{attribute 'no_explicit_call' := 'do not call this function block directly'}
FUNCTION_BLOCK FB_Scalar IMPLEMENTS I_Scalar, I_Addition, I_Subtraction, I_Multiplication, I_Division
VAR
	_fValue : LREAL; 
END_VAR

METHOD DivideBy : I_Division
VAR_INPUT
	ipObject : I_Object;
END_VAR
VAR_OUTPUT
	e : E_OperatorError;
END_VAR
VAR
	Tmp : LREAL;
	ipNumber : I_Scalar;
END_VAR
DivideBy := THIS^;

IF NOT __QUERYINTERFACE(ipObject, ipNumber) THEN e := E_OperatorError.TypeMismatch; RETURN; END_IF

Tmp := ipNumber.ToF64(e => e);
IF Tmp = 0 THEN 
	THIS^._fValue := SEL(Tmp > 0, -1*TO_LREAL('#Inf'), TO_LREAL('#Inf'));
	RETURN;
	END_IF

IF e <> E_OperatorError.NoError THEN 
	THIS^._fValue := ipNumber.ToF64();
	END_IF

THIS^._fValue := THIS^.ToF64() / ipNumber.ToF64();
END_METHOD

{attribute 'hide'}
METHOD FB_init : BOOL
VAR_INPUT
	bInitRetains : BOOL; // if TRUE, the retain variables are initialized (warm start / cold start)
	bInCopyCode : BOOL;  // if TRUE, the instance afterwards gets moved into the copy code (online change)
	fInitValue : LREAL;
END_VAR
THIS^._fValue := fInitValue;
END_METHOD

METHOD Minus : I_Subtraction
VAR_INPUT
	ipObject : I_Object;
END_VAR
VAR_OUTPUT
	e : E_OperatorError;
END_VAR
VAR
	e1, e2 : E_OperatorError;
	ipNumber : I_Scalar;
END_VAR
Minus := THIS^;

IF NOT __QUERYINTERFACE(ipObject, ipNumber) THEN
  e := E_OperatorError.TypeMismatch; 
  RETURN;
  END_IF

THIS^._fValue := THIS^.ToF64(e => e1) - ipNumber.ToF64(e => e2);

e := MAX(e1, e2);
END_METHOD

METHOD Plus : I_Addition
VAR_INPUT
	ipObject : I_Object;
END_VAR
VAR_OUTPUT
	e : E_OperatorError;
END_VAR
VAR
	e1, e2 : E_OperatorError;
	ipNumber : I_Scalar;
END_VAR
Plus := THIS^;

IF NOT __QUERYINTERFACE(ipObject, ipNumber) THEN e := E_OperatorError.TypeMismatch; RETURN; END_IF

THIS^._fValue := THIS^.ToF64(e => e1) + ipNumber.ToF64(e => e2);

e := MAX(e1, e2);
END_METHOD

METHOD SetValue : REFERENCE TO FB_Scalar
VAR_INPUT
	fValue : LREAL;
END_VAR
SetValue REF= THIS^;

THIS^._fValue := fValue;
END_METHOD

METHOD Times : I_Multiplication
VAR_INPUT
	ipObject : I_Object;
END_VAR
VAR_OUTPUT
	e : E_OperatorError;
END_VAR
VAR
	e1, e2 : E_OperatorError;
	ipNumber : I_Scalar;
END_VAR
Times := THIS^;

IF NOT __QUERYINTERFACE(ipObject, ipNumber) THEN e := E_OperatorError.TypeMismatch; RETURN; END_IF

THIS^._fValue := THIS^.ToF64(e => e1) * ipNumber.ToF64( e => e2);

e := MAX(e1, e2);
END_METHOD

METHOD ToF64 : LREAL
VAR_OUTPUT
	e	: E_OperatorError;
END_VAR
ToF64 := THIS^._fValue;

IF TO_STRING(THIS^._fValue) = '#NaN' THEN 
	e := E_OperatorError.NaN;
ELSIF TO_STRING(THIS^._fValue) = '#Inf' THEN
	e := E_OperatorError.PositiveInfinity;
ELSIF TO_STRING(THIS^._fValue) = '-#Inf' THEN
	e := E_OperatorError.NegativeInfinity;
	END_IF
END_METHOD

METHOD ToI64 : LINT
VAR_OUTPUT
	e	: E_OperatorError;
END_VAR
ToI64 := TO_LINT(THIS^._fValue);

// Check for truncation.
IF Tc2_Math.FRAC(THIS^._fValue) <> 0  THEN 
	e := E_OperatorError.Truncation;
	END_IF
END_METHOD

METHOD ToU8 : BYTE
VAR_OUTPUT
	e	: E_OperatorError;
END_VAR
ToU8 := TO_BYTE(THIS^._fValue);

// Check for truncation.
IF Tc2_Math.FRAC(THIS^._fValue) <> 0  THEN 
	e := E_OperatorError.Truncation;
	END_IF

// Bounds check.
IF THIS^._fValue < 0 OR THIS^._fValue > 255 THEN 
	e := E_OperatorError.IntegerOverflow;
	END_IF
END_METHOD

END_FUNCTION_BLOCK

(* stored: Version 1.1.0.1, ProductVersion 3.1.4024.12
   POU FB_Scalar: Id {06260915-57c3-4c39-8ab5-e6a4c7e7c262}, SpecialFunc None
   Folder Constructor: Id {a996651f-3295-46b6-b977-e378ab8cc6d3}
   Folder IOperatorX: Id {fb9cacd6-caa0-492a-82b5-8880a839455e}
   Folder IScalar: Id {3e8f876f-10c8-4aaa-9fa8-9b178ddb88f2}
   Method DivideBy: Id {b0d0123e-cfb1-4101-8e18-a861c0279c74}
   Method FB_init: Id {63985488-ffd6-4997-a4e0-e9bffe3b7aa1}
   Method Minus: Id {18369c4d-9f09-40b4-9308-b820645b5f26}
   Method Plus: Id {60384213-cda5-42bb-a2ed-7a4ea44476e7}
   Method SetValue: Id {1949f961-9b2e-471c-8bbf-54413b825d1c}
   Method Times: Id {2654030e-17b8-414f-9c51-0561518f02d5}
   Method ToF64: Id {b907d5d0-24ee-478b-a026-7a64638e8296}
   Method ToI64: Id {52419fd5-870a-4326-9013-32b165d32938}
   Method ToU8: Id {7391b4cf-f0f6-43c4-80a6-4b323817aa37} *)
